FUNCTION_BLOCK FB_InitPM
VAR_INPUT
	sIpAddress		: STRING;
	nUnitID			: BYTE;
	nPort			: UINT;
END_VAR

VAR_OUTPUT
END_VAR

VAR_IN_OUT
	PM		:	ST_PowerMeter;
END_VAR

VAR
END_VAR

(******** Init Connection **************)
PM.Conn.sIPAddress		:= sIpAddress;
PM.Conn.nUnitID			:= nUnitID;
PM.Conn.nPort			:= nPort;

END_FUNCTION_BLOCK

(* stored: Version 1.1.0.1, ProductVersion 3.1.4024.12
   POU FB_InitPM: Id {3f59bf5b-6dcb-4ed2-9e76-1262f0fb922f}, SpecialFunc None *)
